FUNCTION_BLOCK FB_ALT_2_PUMPS
VAR_INPUT
	LS_1 : BOOL;
	LS_2 : BOOL;
	LS_3 : BOOL;
	LS_4 : BOOL;
END_VAR
VAR_OUTPUT
	Pump_1 : BOOL;
	Pump_2 : BOOL;
END_VAR
VAR
	Reset_pumps: BOOL;
	Alt_pumps: BOOL;
	
	Pump_Count : INT := 0;
	LS_2_Pump_1: BOOL;
	LS_2_Pump_2: BOOL;
	LS_3_Pump_1: BOOL;
	LS_3_Pump_2: BOOL;
END_VAR
VAR // added by the converter: edge detectors and wires of the graphical bodies
    _rt1 : R_TRIG;
    _w1, _w2, _w3 : BOOL;
END_VAR

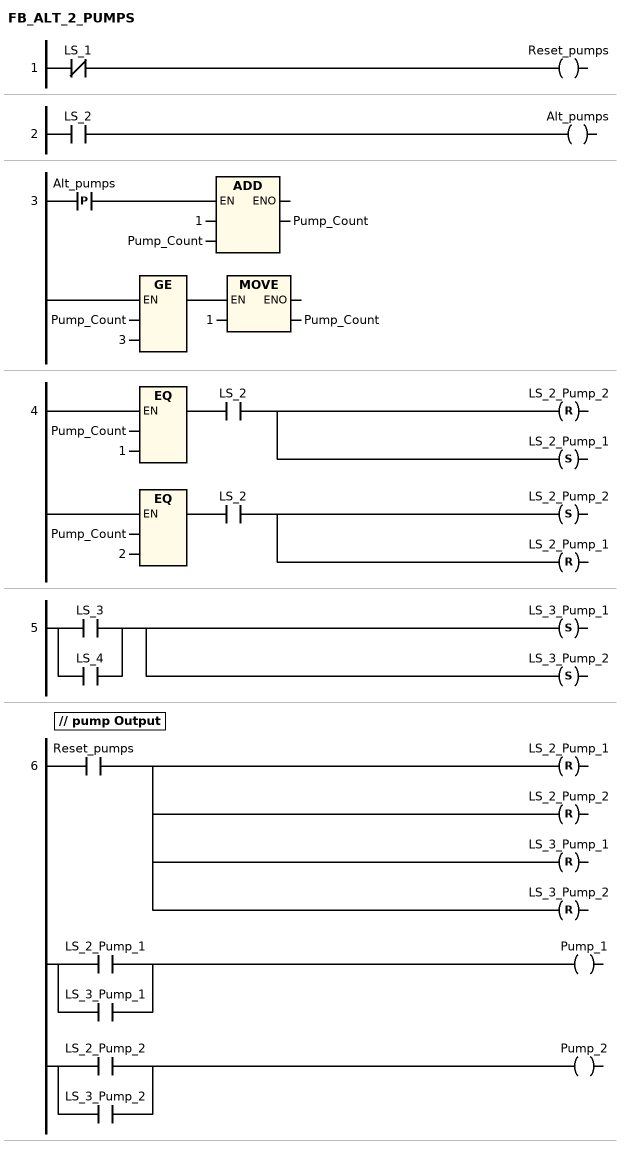
// NETWORK 1
Reset_pumps := NOT LS_1;

// NETWORK 2
Alt_pumps := LS_2;

// NETWORK 3
_rt1(CLK := Alt_pumps);
IF _rt1.Q THEN Pump_Count := 1 + Pump_Count; END_IF
IF Pump_Count >= 3 THEN Pump_Count := 1; END_IF

// NETWORK 4
_w1 := Pump_Count = 1 AND LS_2;
LS_2_Pump_2 R= _w1;
LS_2_Pump_1 S= _w1;
_w2 := Pump_Count = 2 AND LS_2;
LS_2_Pump_2 S= _w2;
LS_2_Pump_1 R= _w2;

// NETWORK 5
_w3 := LS_3 OR LS_4;
LS_3_Pump_1 S= _w3;
LS_3_Pump_2 S= _w3;

// NETWORK 6
// label: // pump Output
LS_2_Pump_1 R= Reset_pumps;
LS_2_Pump_2 R= Reset_pumps;
LS_3_Pump_1 R= Reset_pumps;
LS_3_Pump_2 R= Reset_pumps;
Pump_1 := LS_2_Pump_1 OR LS_3_Pump_1;
Pump_2 := LS_2_Pump_2 OR LS_3_Pump_2;

END_FUNCTION_BLOCK

(* stored: Version 1.1.0.1, ProductVersion 3.1.4024.13
   POU FB_ALT_2_PUMPS: Id {288bbdf7-42c6-4f68-b9d2-50fa102b3fc5}, SpecialFunc None *)
